TYPE DUT_MainlineFixture :
STRUCT
		xMaterialOnOff : BOOL ;
    stProduct : DUT_PartStatus ;
		stProductFlag :DUT_PartFlag;
		stProcessData:DUT_LidChecking;
		arCycletimeStation: ARRAY[1..20] OF REAL;
END_STRUCT
END_TYPE

(* stored: Version 1.1.0.1, ProductVersion 3.1.4024.9
   DUT DUT_MainlineFixture: Id {8707e05e-86c7-4629-a577-967014eadd0d} *)
